FUNCTION fcWriteOutput : REAL
//Writes a scaled output

VAR_INPUT
	rInValue	: REAL;		// Input value
	rInScaledMax	: REAL;		// Engineering units range max
	rInScaledMin	: REAL;		// Engineering units range min
	rInRawMax		: REAL;		// Raw maximum - overflow limit
	rInRawMin		: REAL;		// Raw minimum - underflow limit
END_VAR
VAR
	rTemp			: REAL;		// Temp REAL value
	rRawMax			: REAL;
	rRawMin			: REAL;
	rRawRange		: REAL;
	rScaledRange	: REAL;
	rOutput			: REAL;
	iOutput			: INT;
END_VAR

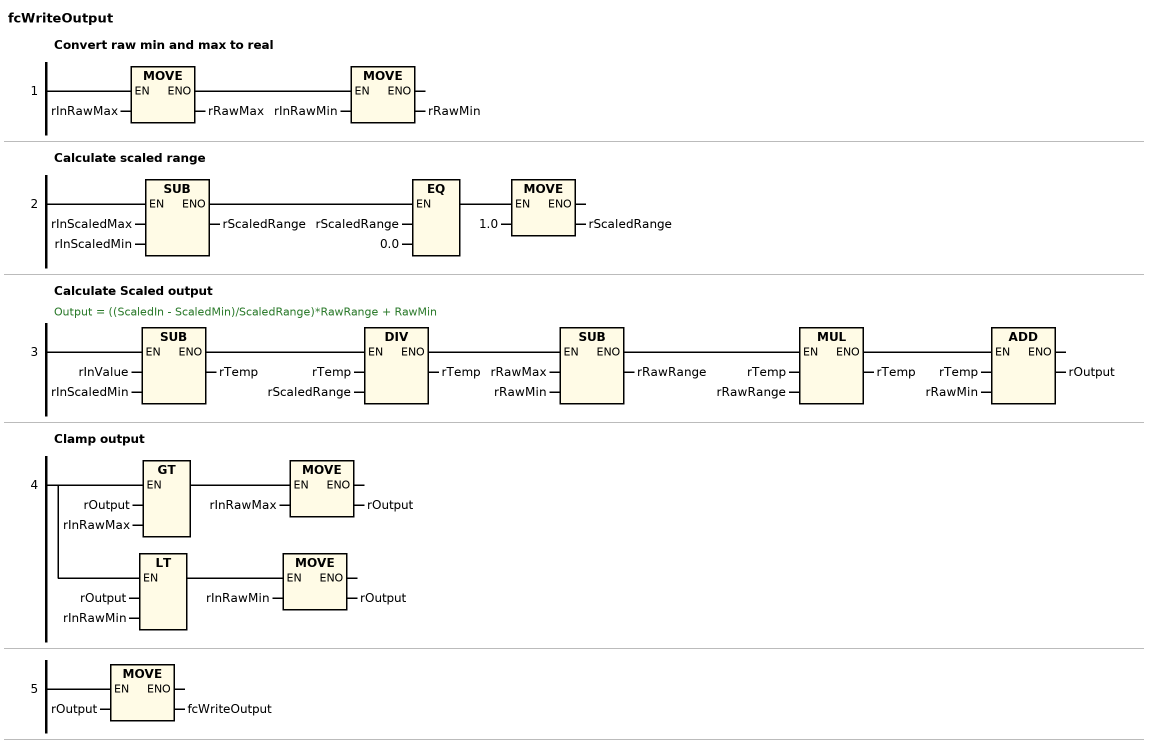
// NETWORK 1: Convert raw min and max to real
rRawMax := rInRawMax;
rRawMin := rInRawMin;

// NETWORK 2: Calculate scaled range
rScaledRange := rInScaledMax - rInScaledMin;
IF rScaledRange = 0.0 THEN rScaledRange := 1.0; END_IF

// NETWORK 3: Calculate Scaled output
// Output = ((ScaledIn - ScaledMin)/ScaledRange)*RawRange + RawMin
rTemp := rInValue - rInScaledMin;
rTemp := rTemp / rScaledRange;
rRawRange := rRawMax - rRawMin;
rTemp := rTemp * rRawRange;
rOutput := rTemp + rRawMin;

// NETWORK 4: Clamp output
IF rOutput > rInRawMax THEN rOutput := rInRawMax; END_IF
IF rOutput < rInRawMin THEN rOutput := rInRawMin; END_IF

// NETWORK 5
fcWriteOutput := rOutput;

END_FUNCTION

(* stored: Version 1.1.0.1, ProductVersion 3.1.4024.12
   POU fcWriteOutput: Id {d030c0d4-dc8e-41b7-8503-243564cdd4d8}, SpecialFunc None *)
